Staubli VAL3: ros_server.pjx

--- ros_server.pjx ---
Parameters version=s7.11 stackSize=5000 millimeterUnit=true
Program file=dataReceiver.pgx
Program file=dataStreamer.pgx
Program file=decodeMsgBody.pgx
Program file=decodeMsgHeader.pgx
Program file=decTrajPt.pgx
Program file=decTrajPtFull.pgx
Program file=encodeAck.pgx
Program file=encodeJState.pgx
Program file=encodeStatus.pgx
Program file=encPrefixHeader.pgx
Program file=encTrajPtAck.pgx
Program file=encTrajPtFAck.pgx
Program file=fetchStatus.pgx
Program file=initParams.pgx
Program file=interpolateVel.pgx
Program file=motionControl.pgx
Program file=pushMotion.pgx
Program file=recvData.pgx
Program file=recvHeartbeat.pgx
Program file=recvMsgBody.pgx
Program file=recvMsgHeader.pgx
Program file=recvTrajPt.pgx
Program file=recvTrajPtFull.pgx
Program file=screenUpdate.pgx
Program file=sendAck.pgx
Program file=sendData.pgx
Program file=sendRosMsg.pgx
Program file=setupRosMsgs.pgx
Program file=start.pgx
Program file=stop.pgx
Program file=toJointArrayRad.pgx
Program file=toJointDeg.pgx
Data file=ros_server.dtx
Library alias=libQueueFuncs path=Disk://ros_libs/QueueFuncs/QueueFuncs.pjx
Library alias=libInterface path=Disk://ros_libs/UserInterface/interfaceDefault/interfaceDefault.pjx autoload=false
Type name=RosSimpleMsg path=Disk://ros_libs/RosSimpleMsg/RosSimpleMsg.pjx
Type name=RobotStatusMsg path=Disk://ros_libs/RobotStatusMsg/RobotStatusMsg.pjx
Type name=JointStateMsg path=Disk://ros_libs/JointStateMsg/JointStateMsg.pjx
Type name=JointTrajPtMsg path=Disk://ros_libs/JointTrajPtMsg/JointTrajPtMsg.pjx
Type name=JointTrajPtFMsg path=Disk://ros_libs/JointTrajPtFMsg/JointTrajPtFMsg.pjx
Type name=JointFbkMsg path=Disk://ros_libs/JointFbkMsg/JointFbkMsg.pjx
Type name=MotionCmd path=Disk://ros_libs/MotionCmd/MotionCmd.pjx
Type name=Header path=Disk://ros_libs/Header/Header.pjx
Type name=Prefix path=Disk://ros_libs/Prefix/Prefix.pjx
Type name=Body path=Disk://ros_libs/Body/Body.pjx
Type name=Queue path=Disk://ros_libs/Queue/Queue.pjx

--- ros_server.dtx ---
public bool bFbkOverrun
public bool bMotionOverrun
public sio siTcpIpFbk = {link=Socket\Feedback}
public sio siTcpIpMotion = {link=Socket\Motion}
public string sStreamTaskName = "publisher"
public string sMotionTaskName
public RosSimpleMsg rosGenericMsg
  [0]
    Header header
      [0]
        num nMsgType
        num nCommType
        num nReplyCode
        num nData[12]
    Prefix prefix
      [0]
        num nLength
        num nData[4]
public tool tTool = {fatherId=flange[0], ioLink=ValveIO\valve1}
public string sTrajPtTaskName
public bool bTrajPtOverrun
public RobotStatusMsg rosStatusMsg
  [0]
    Body body
      [0]
        num nData[28]
    Header header
      [0]
        num nMsgType
        num nCommType
        num nReplyCode
        num nData[12]
    Prefix prefix
      [0]
        num nLength
        num nData[4]
    RobotStatus robotStatus
      [0]
        num nDrivesPowered
        num nEStopped
        num nErrorCode
        num nInError
        num nInMotion
        num nMode
        num nMotionPossible
public JointStateMsg rosJointMsg
  [0]
    Header header
      [0]
        num nMsgType
        num nCommType
        num nReplyCode
        num nData[12]
    Body body
      [0]
        num nData[44]
    JointState jointState
      [0]
        num nSeq
        num nJoints[10]
    Prefix prefix
      [0]
        num nLength
        num nData[4]
public JointTrajPtMsg rosTrajPtMsg
  [0]
    Header header
      [0]
        num nMsgType
        num nCommType
        num nReplyCode
        num nData[12]
    JointTrajPt jointTrajPt
      [0]
        num nSeq
        num nJoints[10]
        num nVelocity
        num nDuration
    Prefix prefix
      [0]
        num nLength
        num nData[4]
    Body body
      [0]
        num nData[52]
public JointTrajPtFMsg rosTrajPtFMsg
  [0]
    Header header
      [0]
        num nMsgType
        num nCommType
        num nReplyCode
        num nData[12]
    Prefix prefix
      [0]
        num nLength
        num nData[4]
    JointTrajPtFull jointTrajPtFull
      [0]
        num nRobotId
        num nSeq
        num nValidFields
        num nTime
        num nPositions[10]
        num nVelocities[10]
        num nAccelerations[10]
    Body body
      [0]
        num nData[136]
public JointFbkMsg rosJointFbkMsg
  [0]
    Header header
      [0]
        num nMsgType
        num nCommType
        num nReplyCode
        num nData[12]
    Prefix prefix
      [0]
        num nLength
        num nData[4]
    JointFeedback jointFeedback
      [0]
        num nRobotId
        num nValidFields
        num nTime
        num nPositions[10]
        num nVelocities[10]
        num nAccelerations[10]
    Body body
      [0]
        num nData[132]
public JointTrajPtFMsg rosTrajPtFAck
  [0]
    Header header
      [0]
        num nMsgType
        num nCommType
        num nReplyCode
        num nData[12]
    Prefix prefix
      [0]
        num nLength
        num nData[4]
    JointTrajPtFull jointTrajPtFull
      [0]
        num nRobotId
        num nSeq
        num nValidFields
        num nTime
        num nPositions[10]
        num nVelocities[10]
        num nAccelerations[10]
    Body body
      [0]
        num nData[136]
public JointTrajPtMsg rosTrajPtAck
  [0]
    Header header
      [0]
        num nMsgType
        num nCommType
        num nReplyCode
        num nData[12]
    JointTrajPt jointTrajPt
      [0]
        num nSeq
        num nJoints[10]
        num nVelocity
        num nDuration
    Prefix prefix
      [0]
        num nLength
        num nData[4]
    Body body
      [0]
        num nData[52]
public bool bScreenOverrun
public string sScreenTaskName
public num nInConnFlag
public num nOutConnFlag
public string sHtbtTaskName
public num nPtsPopped
public bool bStopNow
public num nMotionProgress
public num nMoveId
public num nMovePts
public num nElapsedTime
public num nHeaderTime
public bool bOverwriteVel
public Queue qMoveBuffer
  [0]
    num nPush
    num nPop
    num nElems
    MotionCmd buffer[10]
      [0]
        mdesc mDesc = {leave=0, reach=0}
        num nDuration
        num nSequence
        joint jJoint
      [1]
        mdesc mDesc = {leave=0, reach=0}
        num nDuration
        num nSequence
        joint jJoint
      [2]
        mdesc mDesc = {leave=0, reach=0}
        num nDuration
        num nSequence
        joint jJoint
      [3]
        mdesc mDesc = {leave=0, reach=0}
        num nDuration
        num nSequence
        joint jJoint
      [4]
        mdesc mDesc = {leave=0, reach=0}
        num nDuration
        num nSequence
        joint jJoint
      [5]
        mdesc mDesc = {leave=0, reach=0}
        num nDuration
        num nSequence
        joint jJoint
      [6]
        mdesc mDesc = {leave=0, reach=0}
        num nDuration
        num nSequence
        joint jJoint
      [7]
        mdesc mDesc = {leave=0, reach=0}
        num nDuration
        num nSequence
        joint jJoint
      [8]
        mdesc mDesc = {leave=0, reach=0}
        num nDuration
        num nSequence
        joint jJoint
      [9]
        mdesc mDesc = {leave=0, reach=0}
        num nDuration
        num nSequence
        joint jJoint
public Queue qTrajPtBuffer
  [0]
    num nPush
    num nPop
    num nElems
    MotionCmd buffer[10]
      [0]
        mdesc mDesc = {leave=0, reach=0}
        num nDuration
        num nSequence
        joint jJoint
      [1]
        mdesc mDesc = {leave=0, reach=0}
        num nDuration
        num nSequence
        joint jJoint
      [2]
        mdesc mDesc = {leave=0, reach=0}
        num nDuration
        num nSequence
        joint jJoint
      [3]
        mdesc mDesc = {leave=0, reach=0}
        num nDuration
        num nSequence
        joint jJoint
      [4]
        mdesc mDesc = {leave=0, reach=0}
        num nDuration
        num nSequence
        joint jJoint
      [5]
        mdesc mDesc = {leave=0, reach=0}
        num nDuration
        num nSequence
        joint jJoint
      [6]
        mdesc mDesc = {leave=0, reach=0}
        num nDuration
        num nSequence
        joint jJoint
      [7]
        mdesc mDesc = {leave=0, reach=0}
        num nDuration
        num nSequence
        joint jJoint
      [8]
        mdesc mDesc = {leave=0, reach=0}
        num nDuration
        num nSequence
        joint jJoint
      [9]
        mdesc mDesc = {leave=0, reach=0}
        num nDuration
        num nSequence
        joint jJoint
num nVel[2]
num nStdMsgType{}
  [JOINT_TRAJ_PT] = 11
  [JOINT_TRAJ_PT_FULL] = 14
num nCommType{}
  [SERVICE_REQUEST] = 2
mdesc mNomSpeed
num nRecHeader
num nDecHeader = 1
num nRecBody = 2
num nDecBody = 3
num nPushMotion = 4
num nAck = 5
num nReset

--- start.pgx ---
program start()
  local num l_nFbkPeriod
  local num l_nMotionPeriod
  local num l_nTrajPeriod
  local num l_nScreenUpdate
  local string l_sVersionMajor
  local num l_nVersionMajor
  local bool l_bOkMajor
  local string l_sVersionMinor
  local num l_nVersionMinor
  local bool l_bOkMinor
begin
  // Copyright (c) 2016, Ocado Technology - Robotics Research Team
  //
  // Licensed under the Apache License, Version 2.0 (the "License");
  // you may not use this file except in compliance with the License.
  // You may obtain a copy of the License at
  //
  //     http://www.apache.org/licenses/LICENSE-2.0
  //
  // Unless required by applicable law or agreed to in writing, software
  // distributed under the License is distributed on an "AS IS" BASIS,
  // WITHOUT WARRANTIES OR CONDITIONS OF ANY KIND, either express or implied.
  // See the License for the specific language governing permissions and
  // limitations under the License.


  // Load interface library for CS8 or CS9
  //
  // CS9 handles the UI differently than CS8, requires
  // the UI funtions to be loaded in seperate libraries

  if(mid(getVersion("System"),1,1) == "7")
    // CS8 - VAL 3 rev 7
    // Check for VAL 3 version >= 7.7
    l_sVersionMajor = mid(getVersion("VAL3"),1,1)
    l_sVersionMinor = mid(getVersion("VAL3"),2,1)
    toNum(l_sVersionMajor, l_nVersionMajor, l_bOkMajor)
    toNum(l_sVersionMinor, l_nVersionMinor, l_bOkMinor)
    if(!l_bOkMajor or !l_bOkMinor)
      popUpMsg("Error reading VAL 3 version")
      taskKill("ros_server~")
    endIf
    if( !((l_nVersionMajor == 7) and (l_nVersionMinor >= 7)))
      // VAL 3 version is too old
      popUpMsg("Error: VAL 3 version is < 7.7, socket communication will not work!")
      taskKill("ros_server~")
    endIf
    libInterface:libLoad("ros_libs/UserInterface/interfaceCS8")
  elseIf(mid(getVersion("System"),1,1) == "8")
    // CS9 - VAL 3 rev 8
    libInterface:libLoad("ros_libs/UserInterface/interfaceCS9")
  endIf

  // feedback task will run every 20ms (50Hz)
  l_nFbkPeriod=0.02
  //l_nFbkPeriod = 0.032 // 30Hz
  //l_nFbkPeriod = 0.05  // 20Hz
  //l_nFbkPeriod = 1.0   //  1Hz

  // motion control task will run every 4ms (250Hz)
  l_nMotionPeriod = 0.004
  //l_nMotionPeriod=0.012  // 83Hz
  //l_nMotionPeriod = 0.05 // 20Hz

  // data (trajectory) reception task will run every 4ms (250Hz)
  l_nTrajPeriod = 0.004
  // not in use at the moment
  l_nScreenUpdate = 1.0

  sStreamTaskName = "streamerTask"
  sTrajPtTaskName = "trajPtTask"
  sMotionTaskName = "motionTask"
  sScreenTaskName = "screenTask"
  sHtbtTaskName = "htbtTask"
  sCartTaskName = "cartTask"

  // initialise TCP/IP parameters
  call initParams()
  // setup prefix and header of ROS messages
  call setupRosMsgs()

  // socket connection status flags: initially disconnected
  nInConnFlag = 0
  nOutConnFlag = 0
  nCartConnFlag = 0
  nCartMsgTime = 0

  // flag defining whether velocity to be overwritten to max. vel.
  bOverwriteVel = false

  nPtsPopped = 0
  nMovePts = 0

  // flush buffer of incoming socket
  clearBuffer(siTcpIpMotion)
  // flush buffer of outgoing socket
  clearBuffer(siTcpIpFbk)
  // flush buffer of cartesian socket
  clearBuffer(siTcpIpCart)

  // check if robot is not in emergency stop and wait until estop is reset
  if(esStatus() == 2)
    popUpMsg("Please reset E-Stop")
    wait(esStatus() < 2)
  endIf

  // before anything else, enable power (only works if robot is in remote mode)
  if(!isPowered())
    if(workingMode() >= 4)
      do
        enablePower()
        delay(2)
      until isPowered()
    else
      popUpMsg("Power must be enabled manually")
    endIf
  endIf

  // reset motion, potentially setting a start joint position for calling autoConnect() in the future
  resetMotion()

  // create joint state and robot status streamer task to send data to industrial_robot_client
  taskCreateSync sStreamTaskName, l_nFbkPeriod, bFbkOverrun, dataStreamer()

  // create trajectory point task to receive data from industrial_robot_client
  taskCreateSync sTrajPtTaskName, l_nTrajPeriod, bTrajPtOverrun, dataReceiver()
  //taskCreate sTrajPtTaskName, 100, dataReceiver()

  // create motion task to synchronously apply motion commands to robot
  taskCreateSync sMotionTaskName, l_nMotionPeriod, bMotionOverrun, motionControl()

  // create synchronous task to update screen
  //taskCreateSync sScreenTaskName, l_nScreenUpdate, bScreenOverrun, screenUpdate()
  taskCreate sScreenTaskName, 10, screenUpdate()

  // create asynchronous task to receive heartbeat on port 11002
  taskCreate sHtbtTaskName, 10, recvHeartbeat()

  // create asynchronous task for cartesian socket on port 11001
  taskCreate sCartTaskName, 10, cartReceiver()

end

--- cartReceiver.pgx ---
public program cartReceiver()
  local bool l_bOk
  local num l_nPrefix[4]
  local num l_nHeader[12]
  local num l_nBody[52]
  local num l_nMsgType
  local num l_nPrefixLen
  local num l_nCommType
  local num l_nReplyCode
  local num l_nCartPoseType
  local num l_nPoseData[9]
  local point l_pTarget
begin
  while (true)
    l_bOk = false
    call recvData(siTcpIpCart, l_nPrefix, nCartConnFlag, l_bOk)
    if (l_bOk)
      call recvData(siTcpIpCart, l_nHeader, nCartConnFlag, l_bOk)
    endIf

    if (l_bOk)
      fromBinary(l_nHeader, 4, "-4l", l_nMsgType)

      if(l_nMsgType==nStdMsgType["CART_GET_POSE"])
        call recvData(siTcpIpCart, l_nBody, nCartConnFlag, l_bOk)
        if (l_bOk)
          nCartMsgTime = clock()
          l_pTarget = here(tTool, world)

          l_nPrefixLen = 64
          l_nCartPoseType = nStdMsgType["CART_POSE"]
          l_nCommType = 1
          l_nReplyCode = 1

          toBinary(l_nPrefixLen, 1, "-4l", l_nPrefix)
          toBinary(l_nCartPoseType, 1, "-4l", l_nHeader)
          toBinary(l_nCommType, 1, "-4l", l_nHeader[4])
          toBinary(l_nReplyCode, 1, "-4l", l_nHeader[8])

          l_nPoseData[0] = 0
          l_nPoseData[1] = l_pTarget.trsf.x * 0.001
          l_nPoseData[2] = l_pTarget.trsf.y * 0.001
          l_nPoseData[3] = l_pTarget.trsf.z * 0.001
          l_nPoseData[4] = l_pTarget.trsf.rx
          l_nPoseData[5] = l_pTarget.trsf.ry
          l_nPoseData[6] = l_pTarget.trsf.rz
          l_nPoseData[7] = 0
          l_nPoseData[8] = 0

          toBinary(l_nPoseData[0], 1, "-4l", l_nBody)
          toBinary(l_nPoseData[1], 1, "4.0l", l_nBody[4])
          toBinary(l_nPoseData[2], 1, "4.0l", l_nBody[8])
          toBinary(l_nPoseData[3], 1, "4.0l", l_nBody[12])
          toBinary(l_nPoseData[4], 1, "4.0l", l_nBody[16])
          toBinary(l_nPoseData[5], 1, "4.0l", l_nBody[20])
          toBinary(l_nPoseData[6], 1, "4.0l", l_nBody[24])
          toBinary(l_nPoseData[7], 1, "4.0l", l_nBody[28])
          toBinary(l_nPoseData[8], 1, "4.0l", l_nBody[32])

          call sendData(siTcpIpCart, l_nPrefix, nCartConnFlag)
          call sendData(siTcpIpCart, l_nHeader, nCartConnFlag)
          call sendData(siTcpIpCart, l_nBody, nCartConnFlag)
        endIf
      endIf
    endIf

    delay(0)
  endWhile
end

--- dataStreamer.pgx ---
public program dataStreamer()
  local num l_nThrottle
  local joint l_jCurrPose
begin
  // Copyright (c) 2016, Ocado Technology - Robotics Research Team
  //
  // Licensed under the Apache License, Version 2.0 (the "License");
  // you may not use this file except in compliance with the License.
  // You may obtain a copy of the License at
  //
  //     http://www.apache.org/licenses/LICENSE-2.0
  //
  // Unless required by applicable law or agreed to in writing, software
  // distributed under the License is distributed on an "AS IS" BASIS,
  // WITHOUT WARRANTIES OR CONDITIONS OF ANY KIND, either express or implied.
  // See the License for the specific language governing permissions and
  // limitations under the License.



  l_nThrottle = 0
  while (true)
    // only attempt to send data if flag indicates that connection is established
    if (nOutConnFlag == 1)
      // fetch current joint positions
      l_jCurrPose=herej()
      // encode and send ROS simple_message ID 10: joint state
      call encodeJState(l_jCurrPose)
      call sendRosMsg(siTcpIpFbk, rosJointMsg.prefix, rosJointMsg.header, rosJointMsg.body, nOutConnFlag)

      // send Robot Status messages 5 times slower than Joint State
      if (l_nThrottle == 5)
        // fetch robot status
        call fetchStatus()
        // encode and send ROS simple_message ID 13: robot status
        call encodeStatus()
        call sendRosMsg(siTcpIpFbk, rosStatusMsg.prefix, rosStatusMsg.header, rosStatusMsg.body, nOutConnFlag)
        l_nThrottle = 0
      endIf
      l_nThrottle = l_nThrottle + 1
    else
      delay(0.1)
    endIf

    // sequence task
    delay(0)
  endWhile
end

--- decodeMsgBody.pgx ---
public program decodeMsgBody(num& x_nMsgRecvState)
  local bool l_bFlag
begin
  // Copyright (c) 2016, Ocado Technology - Robotics Research Team
  //
  // Licensed under the Apache License, Version 2.0 (the "License");
  // you may not use this file except in compliance with the License.
  // You may obtain a copy of the License at
  //
  //     http://www.apache.org/licenses/LICENSE-2.0
  //
  // Unless required by applicable law or agreed to in writing, software
  // distributed under the License is distributed on an "AS IS" BASIS,
  // WITHOUT WARRANTIES OR CONDITIONS OF ANY KIND, either express or implied.
  // See the License for the specific language governing permissions and
  // limitations under the License.



  l_bFlag=false

  switch rosGenericMsg.header.nMsgType
    case nStdMsgType["JOINT_TRAJ_PT"]
      call decTrajPt(l_bFlag)
    break
    case nStdMsgType["JOINT_TRAJ_PT_FULL"]
      call decTrajPtFull(l_bFlag)
    break
    default
    break
  endSwitch

  if (l_bFlag == true)
    // move on to state 4: push motion into buffer
    x_nMsgRecvState=nPushMotion
  else
    // error whilst decoding msg body...
    if (rosGenericMsg.header.nCommType==2)
      switch rosGenericMsg.header.nMsgType
        case nStdMsgType["JOINT_TRAJ_PT"]
          rosTrajPtAck.header.nReplyCode=2
        break
        case nStdMsgType["JOINT_TRAJ_PT_FULL"]
          rosTrajPtFAck.header.nReplyCode=2
        break
        default
        break
      endSwitch
      // jump to state 5: sendAck()
      x_nMsgRecvState=nAck
    else
      // reset state machine, since no ACK is required
      x_nMsgRecvState=nReset
    endIf
  endIf
end

--- encodeJState.pgx ---
public program encodeJState(joint& x_jCurrPose)
begin
  // Copyright (c) 2016, Ocado Technology - Robotics Research Team
  //
  // Licensed under the Apache License, Version 2.0 (the "License");
  // you may not use this file except in compliance with the License.
  // You may obtain a copy of the License at
  //
  //     http://www.apache.org/licenses/LICENSE-2.0
  //
  // Unless required by applicable law or agreed to in writing, software
  // distributed under the License is distributed on an "AS IS" BASIS,
  // WITHOUT WARRANTIES OR CONDITIONS OF ANY KIND, either express or implied.
  // See the License for the specific language governing permissions and
  // limitations under the License.



  // encode 'prefix' and 'header'
  call encPrefixHeader(rosJointMsg.prefix, rosJointMsg.header)

  // encode 'sequence' variable of body message (data)
  toBinary(rosJointMsg.jointState.nSeq,1,"-4l",rosJointMsg.body.nData)

  call toJointArrayRad(x_jCurrPose, rosJointMsg.jointState.nJoints)

  // encode 10 values representing joints[10]
  toBinary(rosJointMsg.jointState.nJoints,10,"4.0l",rosJointMsg.body.nData[4])
end

--- initParams.pgx ---
public program initParams()
  local num l_nRetVal
begin
  // Copyright (c) 2016, Ocado Technology - Robotics Research Team
  //
  // Licensed under the Apache License, Version 2.0 (the "License");
  // you may not use this file except in compliance with the License.
  // You may obtain a copy of the License at
  //
  //     http://www.apache.org/licenses/LICENSE-2.0
  //
  // Unless required by applicable law or agreed to in writing, software
  // distributed under the License is distributed on an "AS IS" BASIS,
  // WITHOUT WARRANTIES OR CONDITIONS OF ANY KIND, either express or implied.
  // See the License for the specific language governing permissions and
  // limitations under the License.



  l_nRetVal=sioCtrl(siTcpIpMotion,"timeout",-1)
  if (l_nRetVal!=0)
    popUpMsg("Error while setting consumer timeout")
  endIf

  l_nRetVal=sioCtrl(siTcpIpFbk,"timeout",-1)
  if (l_nRetVal!=0)
    popUpMsg("Error while setting producer timeout")
  endIf

  l_nRetVal=sioCtrl(siTcpIpCart,"timeout",-1)
  if (l_nRetVal!=0)
    popUpMsg("Error while setting cartesian timeout")
  endIf
end

--- motionControl.pgx ---
public program motionControl()
  local MotionCmd l_mTrajPt
  local bool l_bFlag
  local MotionCmd l_motion
  local num l_nElems
begin
  // Copyright (c) 2016, Ocado Technology - Robotics Research Team
  //
  // Licensed under the Apache License, Version 2.0 (the "License");
  // you may not use this file except in compliance with the License.
  // You may obtain a copy of the License at
  //
  //     http://www.apache.org/licenses/LICENSE-2.0
  //
  // Unless required by applicable law or agreed to in writing, software
  // distributed under the License is distributed on an "AS IS" BASIS,
  // WITHOUT WARRANTIES OR CONDITIONS OF ANY KIND, either express or implied.
  // See the License for the specific language governing permissions and
  // limitations under the License.



  nMoveId = -1

  while(true)
    // check connection status, and whether to stop motion
    if(nInConnFlag == 1 and nOutConnFlag == 1 and bStopNow == false)

      // process trajectory point from trajectory buffer
      call libQueueFuncs:getNumElems(qTrajPtBuffer, l_nElems)
      if(l_nElems > 0)
        call libQueueFuncs:pop(qTrajPtBuffer,l_mTrajPt, l_bFlag)
        if(l_bFlag == true)
          nPtsPopped = nPtsPopped + 1
          call libQueueFuncs:push(qMoveBuffer,l_mTrajPt,l_bFlag)
        endIf
      endIf

      // process motion command from move buffer
      // @TODO move buffer should have elements previously interpolated to ensure they are 4 ms apart
      call libQueueFuncs:getNumElems(qMoveBuffer, l_nElems)
      if(l_nElems > 0)
        call libQueueFuncs:pop(qMoveBuffer,l_motion,l_bFlag)
        if(l_bFlag == true)
          nMovePts = nMovePts + 1

          // Velocity buffer to smooth out last traj point
          nVel[1] = nVel[0]
          nVel[0] = rosTrajPtMsg.jointTrajPt.nVelocity

          // Interpolate velocity for last point in trajectory
          call interpolateVel(l_motion)

          // contrary to what we did earlier, we unconditionally add the traj pt to the motion queue:
          // there doesn't appear to be a way to compare the 'current pose' of the robot to the pts
          // in the trajectory at the appropriate time (ie: when the robot is in motion and about to
          // start executing the segment towards 'l_motion').
          // Checking for dist(l_motion, herej()) (pseudo code) would not be correct as there will
          // always be a delay in the data coming out of herej() and the actual pose of the robot.
          // @TODO potentially set move id according to sequence value
          nMoveId = movej(l_motion.jJoint, tTool, l_motion.mDesc)
        endIf
      endIf
    else
      // stop immediately -- resetMotion() also resets moveId
      resetMotion()
      // clear buffers
      call libQueueFuncs:clear(qTrajPtBuffer)
      call libQueueFuncs:clear(qMoveBuffer)
      bStopNow = false

      // debug
      nPtsPopped = 0
      nMovePts = 0
    endIf

    nMotionProgress = getMoveId()

    // sequence task
    delay(0)
  endWhile
end

--- pushMotion.pgx ---
public program pushMotion(num& x_nMsgRecvState)
  local bool l_bOk
  local num l_nCounter
  local num l_nJointError
  local MotionCmd l_mTrajPt
begin
  // Copyright (c) 2016, Ocado Technology - Robotics Research Team
  //
  // Licensed under the Apache License, Version 2.0 (the "License");
  // you may not use this file except in compliance with the License.
  // You may obtain a copy of the License at
  //
  //     http://www.apache.org/licenses/LICENSE-2.0
  //
  // Unless required by applicable law or agreed to in writing, software
  // distributed under the License is distributed on an "AS IS" BASIS,
  // WITHOUT WARRANTIES OR CONDITIONS OF ANY KIND, either express or implied.
  // See the License for the specific language governing permissions and
  // limitations under the License.



  switch rosGenericMsg.header.nMsgType
    case nStdMsgType["JOINT_TRAJ_PT"]
      l_mTrajPt.nSequence=rosTrajPtMsg.jointTrajPt.nSeq

      // ROS positions are SI units; convert to controller-native units
      // (j1..j3: rad->deg, j4: m->mm)
      call toJointDeg(rosTrajPtMsg.jointTrajPt.nJoints, l_mTrajPt.jJoint)

      // from industrial_robot_client/src/joint_trajectory_interface.cpp
      // JointTrajectoryInterface::trajectory_to_msgs()
      // JointTrajectoryInterface::calc_speed()
      // velocity is converted to a scalar value representing % of max velocity,
      // such that 0.2 = 20% of maximum joint speed
      l_mTrajPt.mDesc.vel= limit((rosTrajPtMsg.jointTrajPt.nVelocity * 100), 0, 100)
      l_mTrajPt.nDuration=rosTrajPtMsg.jointTrajPt.nDuration

    break
    case nStdMsgType["JOINT_TRAJ_PT_FULL"]
      l_mTrajPt.nSequence=rosTrajPtFMsg.jointTrajPtFull.nSeq
      l_mTrajPt.nDuration=rosTrajPtFMsg.jointTrajPtFull.nTime

      // ROS positions are SI units; convert to controller-native units
      // (j1..j3: rad->deg, j4: m->mm)
      call toJointDeg(rosTrajPtFMsg.jointTrajPtFull.nPositions, l_mTrajPt.jJoint)

      // from industrial_robot_client/src/joint_trajectory_interface.cpp
      // JointTrajectoryInterface::trajectory_to_msgs()
      // JointTrajectoryInterface::calc_speed()
      // velocity is converted to a scalar value representing % of max velocity,
      // such that 0.2 = 20% of maximum joint speed
      l_mTrajPt.mDesc.vel= limit((rosTrajPtFMsg.jointTrajPtFull.nVelocities[0] * 100), 0, 100)
      // not sure about accelerations as yet
      l_mTrajPt.mDesc.accel=rosTrajPtFMsg.jointTrajPtFull.nAccelerations[0]
      l_mTrajPt.mDesc.decel=l_mTrajPt.mDesc.accel
    break
    default
    break
  endSwitch

  // see github.com/ros-industrial/industrial_core/simple_message/include/simple_message/joint_traj_pt.h
  if(l_mTrajPt.nSequence==-4)
    // set flag to stop immediately
    bStopNow=true
  else
    // check whether velocity value should be overwritten with value set on teach pendant
    if(bOverwriteVel == true)
      // overwrite velocity (and acceleration - ?)
      //l_mTrajPt.mDesc.vel = getMonitorSpeed()
      // explicitly setting accel and decel to VAL3 default values
      l_mTrajPt.mDesc.accel = mNomSpeed.accel
      l_mTrajPt.mDesc.decel = mNomSpeed.decel
    endIf
    // only push motion into buffer if not a STOP message
    // and if joint positions are within software joint limits
    // and if velocity is greater than zero (beucase movej() will not accept vel <= 0)
    if(isInRange(l_mTrajPt.jJoint) and l_mTrajPt.mDesc.vel > 0)
      call libQueueFuncs:push(qTrajPtBuffer,l_mTrajPt,l_bOk)
    else
      l_bOk = false
    endIf

    if(l_bOk==false)
      // could not push trajectory point into buffer
      // thus ACK should flag FAILURE, but only if comm type is request
      if(rosGenericMsg.header.nCommType==nCommType["SERVICE_REQUEST"])
        switch rosGenericMsg.header.nMsgType
          case nStdMsgType["JOINT_TRAJ_PT"]
            rosTrajPtAck.header.nReplyCode=2
          break
          case nStdMsgType["JOINT_TRAJ_PT_FULL"]
            rosTrajPtFAck.header.nReplyCode=2
          break
          default
          break
        endSwitch
      endIf
    endIf
  endIf
  // check whether ACK should be sent
  if(rosGenericMsg.header.nCommType == nCommType["SERVICE_REQUEST"])
    // comm type request requires ACK
    x_nMsgRecvState = nAck
  else
    // other comm types (e.g., topic) does not require ACK, hence skip state
    x_nMsgRecvState = nReset
  endIf
end

--- recvMsgBody.pgx ---
public program recvMsgBody(num& x_nMsgRecvState)
  local bool l_bFlag
begin
  // Copyright (c) 2016, Ocado Technology - Robotics Research Team
  //
  // Licensed under the Apache License, Version 2.0 (the "License");
  // you may not use this file except in compliance with the License.
  // You may obtain a copy of the License at
  //
  //     http://www.apache.org/licenses/LICENSE-2.0
  //
  // Unless required by applicable law or agreed to in writing, software
  // distributed under the License is distributed on an "AS IS" BASIS,
  // WITHOUT WARRANTIES OR CONDITIONS OF ANY KIND, either express or implied.
  // See the License for the specific language governing permissions and
  // limitations under the License.



  l_bFlag=false

  switch rosGenericMsg.header.nMsgType
    case nStdMsgType["JOINT_TRAJ_PT"]
      call recvTrajPt(l_bFlag)
    break
    case nStdMsgType["JOINT_TRAJ_PT_FULL"]
      call recvTrajPtFull(l_bFlag)
    break
    default
    break
  endSwitch

  if (l_bFlag == true)
    // move on to state 3: decode msg body
    x_nMsgRecvState=nDecBody
  else
    // error whilst receiving msg body, reset state machine
    x_nMsgRecvState=nReset
  endIf
end

--- screenUpdate.pgx ---
public program screenUpdate()
  local num l_nKey
  local num l_nExecStatus
  local num l_nElems
  local num l_nCartMsgAge
begin
  // Copyright (c) 2016, Ocado Technology - Robotics Research Team
  //
  // Licensed under the Apache License, Version 2.0 (the "License");
  // you may not use this file except in compliance with the License.
  // You may obtain a copy of the License at
  //
  //     http://www.apache.org/licenses/LICENSE-2.0
  //
  // Unless required by applicable law or agreed to in writing, software
  // distributed under the License is distributed on an "AS IS" BASIS,
  // WITHOUT WARRANTIES OR CONDITIONS OF ANY KIND, either express or implied.
  // See the License for the specific language governing permissions and
  // limitations under the License.

  l_nExecStatus = 0

  call libInterface:init()

  while(true)

    // clear screen
    call libInterface:clearScreen()

    // @TODO: Remove all code related to velocity overwrite
    //    // toggle velocity overwrite upon release of F1 key
    //    l_nKey = getKey(scMonitor)
    //    call libQueueFuncs:getNumElems(qMoveBuffer,l_nElems)
    //    if (l_nKey == 277 and bOverwriteVel == false)
    //      if (l_nElems == 0)
    //        bOverwriteVel = true
    //      else
    //        popUpMsg("Motion buffer not empty; cannot enable V/OW")
    //      endIf
    //    elseIf (l_nKey == 278 and bOverwriteVel == true)
    //      if (l_nElems == 0)
    //        bOverwriteVel = false
    //      else
    //        popUpMsg("Motion buffer not empty; cannot disable V/OW")
    //      endIf
    //    endIf

    // update connection status on port 11000
    call libInterface:motionStatus(nInConnFlag)

    // update cartesian status on port 11001
    if (nCartMsgTime > 0)
      l_nCartMsgAge = clock() - nCartMsgTime
    else
      l_nCartMsgAge = -1
    endIf
    call libInterface:cartStatus(nCartConnFlag, l_nCartMsgAge)

    // update connection status on port 11002
    call libInterface:feedbackStatus(nOutConnFlag)

    // update trajectory buffer size
    call libQueueFuncs:getNumElems(qTrajPtBuffer,l_nElems)
    call libInterface:trajBuffer(l_nElems,nPtsPopped)

    // do the same for move buffer
    call libQueueFuncs:getNumElems(qMoveBuffer,l_nElems)
    call libInterface:motionBuffer(l_nElems,nPtsPopped)

    // display velocity overwrite status
    call libInterface:velOverwrite(bOverwriteVel)

    // display nMoveId and nMotionProgress
    call libInterface:motionProgress(nMoveId,nMotionProgress)

    // display time between valid trajectory point received and ACK sent
    call libInterface:ack(nHeaderTime,nElapsedTime)

    // update debug status
    call libInterface:debug(l_nExecStatus)

    //    // add Function keys labels
    //    gotoxy(scMonitor, 30,13)
    //    put(scMonitor, "V/ON")
    //    gotoxy(scMonitor, 35,13)
    //    put(scMonitor, "V/OFF")

    // sequence task
    //delay(0)
    delay(0.5)
  endWhile
end

--- toJointArrayRad.pgx ---
public program toJointArrayRad(joint& x_jJoint, num& x_nJointArray[])
  local num l_nDeg2Rad
  local num l_nMm2M
begin
  // Copyright (c) 2016, Ocado Technology - Robotics Research Team
  //
  // Licensed under the Apache License, Version 2.0 (the "License");
  // you may not use this file except in compliance with the License.
  // You may obtain a copy of the License at
  //
  //     http://www.apache.org/licenses/LICENSE-2.0
  //
  // Unless required by applicable law or agreed to in writing, software
  // distributed under the License is distributed on an "AS IS" BASIS,
  // WITHOUT WARRANTIES OR CONDITIONS OF ANY KIND, either express or implied.
  // See the License for the specific language governing permissions and
  // limitations under the License.



  l_nDeg2Rad = 0.01745329251
  l_nMm2M = 0.001

  // RS60 mapping: j1, j2, j4 are revolute (deg->rad),
  // j3 is prismatic (mm->m).
  x_nJointArray[0] = x_jJoint.j1 * l_nDeg2Rad
  x_nJointArray[1] = x_jJoint.j2 * l_nDeg2Rad
  x_nJointArray[2] = x_jJoint.j3 * l_nMm2M
  x_nJointArray[3] = x_jJoint.j4 * l_nDeg2Rad
  x_nJointArray[4] = 0
  x_nJointArray[5] = 0
end

--- toJointDeg.pgx ---
public program toJointDeg(num& x_nJointArray[], joint& x_jJoint)
  local num l_nRad2Deg
  local num l_nM2Mm
begin
  // Copyright (c) 2016, Ocado Technology - Robotics Research Team
  //
  // Licensed under the Apache License, Version 2.0 (the "License");
  // you may not use this file except in compliance with the License.
  // You may obtain a copy of the License at
  //
  //     http://www.apache.org/licenses/LICENSE-2.0
  //
  // Unless required by applicable law or agreed to in writing, software
  // distributed under the License is distributed on an "AS IS" BASIS,
  // WITHOUT WARRANTIES OR CONDITIONS OF ANY KIND, either express or implied.
  // See the License for the specific language governing permissions and
  // limitations under the License.



  l_nRad2Deg = 57.2957795131
  l_nM2Mm = 1000

  // RS60/RS-TS-safe mapping: first three axes are revolute (rad->deg),
  // fourth axis is linear (m->mm).
  x_jJoint.j1 = x_nJointArray[0] * l_nRad2Deg
  x_jJoint.j2 = x_nJointArray[1] * l_nRad2Deg
  x_jJoint.j3 = x_nJointArray[2] * l_nRad2Deg
  x_jJoint.j4 = x_nJointArray[3] * l_nM2Mm
end

--- toJointRxDeg.pgx ---
public program toJointRxDeg(num& x_nJointArray[], joint& x_jJoint)
  local num l_nRad2Deg
  local num l_nM2Mm
begin
  // Copyright (c) 2016, Ocado Technology - Robotics Research Team
  //
  // Licensed under the Apache License, Version 2.0 (the "License");
  // you may not use this file except in compliance with the License.
  // You may obtain a copy of the License at
  //
  //     http://www.apache.org/licenses/LICENSE-2.0
  //
  // Unless required by applicable law or agreed to in writing, software
  // distributed under the License is distributed on an "AS IS" BASIS,
  // WITHOUT WARRANTIES OR CONDITIONS OF ANY KIND, either express or implied.
  // See the License for the specific language governing permissions and
  // limitations under the License.



  l_nRad2Deg = 57.2957795131
  l_nM2Mm = 1000

  // RS60/RS-TS-safe mapping: first three axes are revolute (rad->deg),
  // fourth axis is linear (m->mm).
  x_jJoint.j1 = x_nJointArray[0] * l_nRad2Deg
  x_jJoint.j2 = x_nJointArray[1] * l_nRad2Deg
  x_jJoint.j3 = x_nJointArray[2] * l_nRad2Deg
  x_jJoint.j4 = x_nJointArray[3] * l_nM2Mm
end
